FUNCTION_BLOCK FB_TestSuite1 EXTENDS FB_TestSuite
VAR_INPUT
END_VAR
VAR_OUTPUT
END_VAR
VAR
END_VAR

TestCaseLongRunning();

METHOD TestCaseLongRunning
VAR_INPUT
END_VAR
TEST('TestCaseLongRunning');

// Test never finishes
//AssertTrue(2+2=4, 'Condition is not true');
//TEST_FINISHED();
END_METHOD

END_FUNCTION_BLOCK

(* stored: Version 1.1.0.1, ProductVersion 3.1.4024.12
   POU FB_TestSuite1: Id {a5ea8811-5301-4f6c-aafd-b2e96e83b4a4}, SpecialFunc None
   Method TestCaseLongRunning: Id {976e0437-3cd7-4f7e-af64-671bf9c25b18} *)
